# EPICS autosave request: measCompApp/Db/measCompVoltageIn_settings.req
$(P)$(R)Range
$(P)$(R).LOPR
$(P)$(R).HOPR
$(P)$(R).PREC
$(P)$(R).SCAN
